FUNCTION MakeRequest : ST_Request
VAR_INPUT
	sTimeInput: STRING;
	stTargetColor: ST_LED;
END_VAR
VAR_OUTPUT
	stOutputRequest: ST_Request;
END_VAR

stOutputRequest.stTargetLED := stTargetColor;

IF len(sTimeInput) = 0 THEN 
	stOutputRequest.tTargetTime := T#3S; 
	stOutputRequest.exists := TRUE;
ELSE 
	stOutputRequest.tTargetTime := STRING_TO_TIME(sTimeInput);
	stOutputRequest.exists := TRUE;
END_IF

END_FUNCTION

(* stored: Version 1.1.0.1, ProductVersion 3.1.4022.12
   POU MakeRequest: Id {7bd72082-ff9a-41aa-8a8b-fa748058917e}, SpecialFunc None *)
